TYPE Person :
STRUCT
	FirstName : STRING;
	LastName : STRING;
	Age : INT;
	Birthday : DATE;
	BirthTown : STRING;
END_STRUCT
END_TYPE

(* stored: Version 1.1.0.1, ProductVersion 3.1.4024.9
   DUT Person: Id {4ab22ee1-9504-0cf2-1eb2-504ac9ed7795} *)
